RoboDK station: pick_and_place.rdk

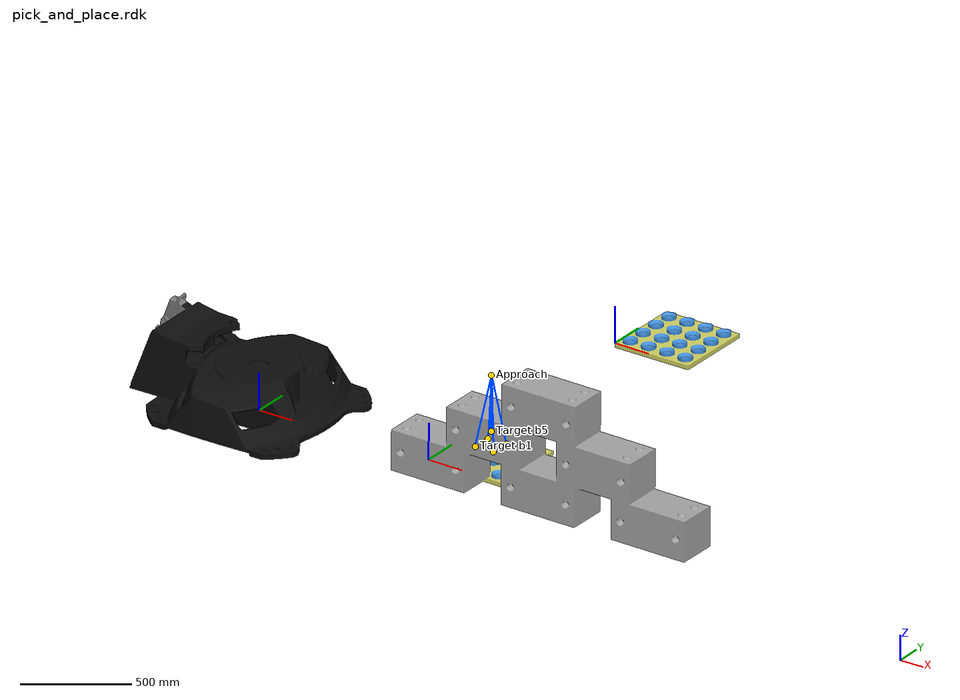
[picture v0: the station drawn from its stored meshes, robots at their saved joint values, targets as dots, program paths as lines]
Station pick_and_place (saved by RoboDK 5.4.1). Poses are relative to the parent item; angles as X-Y-Z fixed-axis rotations.
  - frame KUKA KR 210 R2700 prime Base at (0, 0, 0) mm
    - robot KUKA KR 210 R2700 prime: 6 axes, payload 210 kg, reach 2696 mm, repeatability 0.06 mm, weight 1111 kg
        joint limits [-185, -140, -120, -350, -122.5, -350] to [185, -5, 155, 350, 122.5, 350]; home [0, -90, 90, 0, 0, 0]; saved at [-155.878, -139.601, -76.488, 37.573, 42.083, 150.477]
      - tool Tool, TCP at (125, 0, 100) mm, rotated rx 0 ry 90 rz 0 deg, size 184.7 x 197.7 x 137.7 mm
    - frame Table 1 at (1500, -821.06, 500) mm, rotated rx 0 ry 0.47 rz 0 deg
      - target Approach (Cartesian target) at (200, 200, 400) mm, rotated rx -180 ry 0 rz -180 deg; joints [-42.973, 13.47, -8.834, -85.041, -43.174, 83.215] of KUKA KR 210 R2700 prime
      - target Target b1 (Cartesian target) at (150, 150, 50) mm, rotated rx -180 ry 0 rz -180 deg; joints [-47.421, 23.634, 13.122, -61.195, -57.174, 44.592] of KUKA KR 210 R2700 prime
      - target Target b2 (Cartesian target) at (250, 150, 50) mm, rotated rx -180 ry 0 rz 180 deg; joints [-43.119, 28.404, 5.363, 120.692, 52.642, -134.368] of KUKA KR 210 R2700 prime
      - target Target b3 (Cartesian target) at (150, 250, 50) mm, rotated rx -180 ry 0 rz 180 deg; joints [-42.803, 18.858, 20.461, 124.38, 55.416, -140.321] of KUKA KR 210 R2700 prime
      - target Target b4 (Cartesian target) at (250, 250, 50) mm, rotated rx -180 ry 0 rz 180 deg; joints [-38.55, 23.97, 12.589, 126.778, 51.084, -139.956] of KUKA KR 210 R2700 prime
      - target Target b5 (Cartesian target) at (200, 200, 120.71) mm, rotated rx -180 ry 0 rz 180 deg; joints [-42.973, 109.891, -190.02, 43.4, 82.794, -6.764] of KUKA KR 210 R2700 prime
      - object brick1 at (0, 0, 0) mm, size 400 x 200 x 210 mm, geometry from brick.stp
      - object brick2 at (600, 0, 0) mm, size 400 x 200 x 210 mm, geometry from brick.stp
      - object base at (0, 0, 0) mm, size 400 x 400 x 34.3 mm
      - object brick3 at (1200, 0, 0) mm, size 400 x 200 x 210 mm, geometry from brick.stp
      - object brick4 at (300, 0, 200) mm, size 400 x 200 x 210 mm, geometry from brick.stp
        - object brick5 at (300, 0, 200) mm, size 400 x 200 x 210 mm, geometry from brick.stp
      - object bric6 at (900, 0, 200) mm, size 400 x 200 x 210 mm, geometry from brick.stp
    - frame Table 2 at (1500, 630.03, 500) mm
      - object base at (0, 0, 0) mm, size 400 x 400 x 34.3 mm
  - program Pick and place (63 instructions, listed below)
  - program Replace objects (1 instructions, listed below)
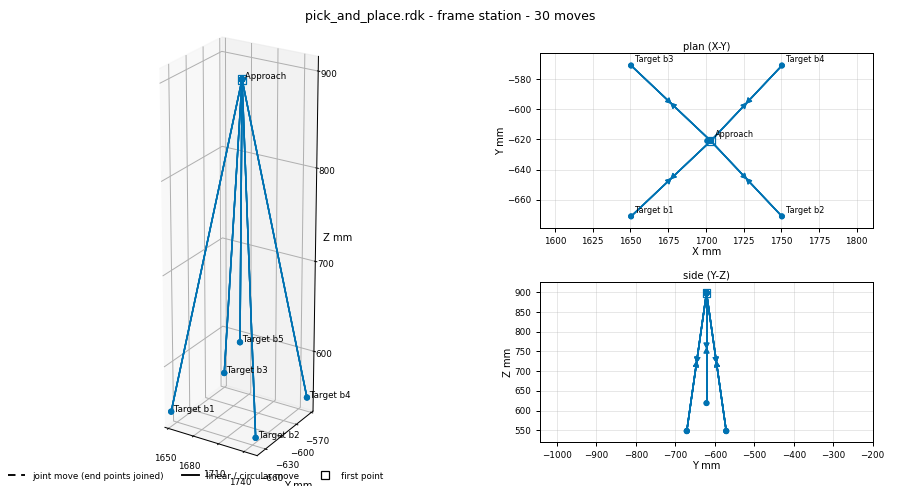
[picture p0: tool path of pick_and_place.rdk in frame station, 30 of 30 moves have a stored position in this frame; points joined in program order, loops and branches not executed]

--- program Pick and place (robot KUKA KR 210 R2700 prime) ---
  Set Frame: Table 1
  Set Tool: Tool
  MoveJ (Approach)
  MoveL (Target b5)
  Attach to Tool
  Call AirValve_On
  MoveL (Approach)
  Set Frame: Table 2
  MoveJ (Approach)
  MoveL (Target b1)
  Detach from Tool
  Call AirValve_Off
  MoveL (Approach)
  Set Frame: Table 1
  MoveJ (Approach)
  MoveL (Target b4)
  Attach to Tool
  Call AirValve_On
  MoveL (Approach)
  Set Frame: Table 2
  MoveJ (Approach)
  MoveL (Target b2)
  Detach from Tool
  Call AirValve_Off
  MoveL (Approach)
  Set Frame: Table 1
  MoveJ (Approach)
  MoveL (Target b3)
  Attach to Tool
  Call AirValve_On
  MoveL (Approach)
  Set Frame: Table 2
  MoveJ (Approach)
  MoveL (Target b3)
  Detach from Tool
  Call AirValve_Off
  MoveL (Approach)
  Set Frame: Table 1
  MoveJ (Approach)
  MoveL (Target b2)
  Attach to Tool
  Call AirValve_On
  MoveL (Approach)
  Set Frame: Table 2
  MoveJ (Approach)
  MoveL (Target b4)
  Detach from Tool
  Call AirValve_Off
  MoveL (Approach)
  Set Frame: Table 1
  MoveJ (Approach)
  MoveL (Target b1)
  Attach to Tool
  Call AirValve_On
  MoveL (Approach)
  Set Frame: Delivery table -> Table 2
  MoveJ (Approach)
  MoveL (Target b5)
  Detach from Tool
  Call AirValve_Off
  MoveL (Approach)
  Pause 5000 ms
  Call Replace objects

--- program Replace objects (robot KUKA KR 210 R2700 prime) ---
  Replace objects
